// TIA Portal V20 export
VAR_GLOBAL   // PLC tag table "Default tag table_4"
END_VAR
